(* CODESYS project export.export

Project tree, tasks and I/O mapping:
  UserGlobals/
    global variables Globals
  UserTypes/
    data type TestTypes
  function SafeInvert [ST]
*)

// UserTypes/TestTypes
TYPE
    TestStruct : STRUCT
        Value   : INT := 0;
        IsValid : BOOL := FALSE;
        Name    : STRING := '';
    END_STRUCT;

    TestEnum : (
        stIdle   := 0,
        stactive := 1,
        stError  := 2
    );
END_TYPE

// UserGlobals/Globals
VAR_GLOBAL
    G_SafeInvertTest : INT := 0;
END_VAR

// SafeInvert
// SafeInvert – merkinvaihto ilman ylivuotoa
//
// INT: alue -32768 .. 32767
// SafeInvert(-32768) = 32767  (rajataan ylärajaan, koska 32768 ylivuotaisi)
// Kaikki muut arvot: tulos = -arvo (normaali negaatio).

FUNCTION SafeInvert : INT
VAR_INPUT
    value : INT;
END_VAR

IF value = -32768 THEN
    SafeInvert := 32767;
ELSE
    SafeInvert := 0 - value;
END_IF;

END_FUNCTION
